FUNCTION_BLOCK SUBLLP0 (* Eight-variable logic proxy to local Subscriber with interface of the globl one *)
  (* Standard: 61499-2 *)
  (* Version 0.0, 2002-11-12, VVV, MLU *)
  (* Compiler header: package fb.rt.net; *)
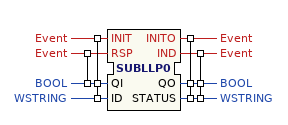
  EVENT_INPUT
    INIT WITH QI, ID; (* Service Initialization *)
    RSP WITH QI; (* Service Response *)
  END_EVENT
  EVENT_OUTPUT
    INITO WITH QO, STATUS; (* Initialization Confirm *)
    IND WITH QO, STATUS; (* Service Indication *)
  END_EVENT
  VAR_INPUT
    QI : BOOL; (* Event Input Qualifier *)
    ID : WSTRING; (* Connection Identifier *)
  END_VAR
  VAR_OUTPUT
    QO : BOOL; (* Event Output Qualifier *)
    STATUS : WSTRING; (* Service Status *)
  END_VAR
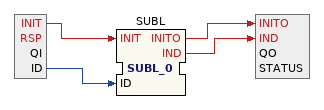
  FBS
    SUBL : SUBL_0;
  END_FBS
  EVENT_CONNECTIONS
    INIT TO SUBL.INIT;
    SUBL.INITO TO INITO;
    SUBL.IND TO IND;
  END_CONNECTIONS
  DATA_CONNECTIONS
    ID TO SUBL.ID;
  END_CONNECTIONS
END_FUNCTION_BLOCK
